FUNCTION_BLOCK FB_AV
VAR_INPUT
END_VAR
VAR_OUTPUT
END_VAR
VAR
	System_Druckluftkompressor_951			: FB_System_DLK_951;
	System_HybriderEnergiespeicher_991		: FB_System_HES_991;
	System_Maschinenversorgung_KW_100		: FB_System_MVKW_100;
	System_Maschinenversorgung_HW_300		: FB_System_MVHW_300;
	System_Haerteofen_961					: FB_System_HO_961;
	System_Maschinenversorgung_WW_245		: FB_System_MVWW_245;
END_VAR
VAR // added by the converter: edge detectors and wires of the graphical bodies
    _w1 : ANY;
END_VAR

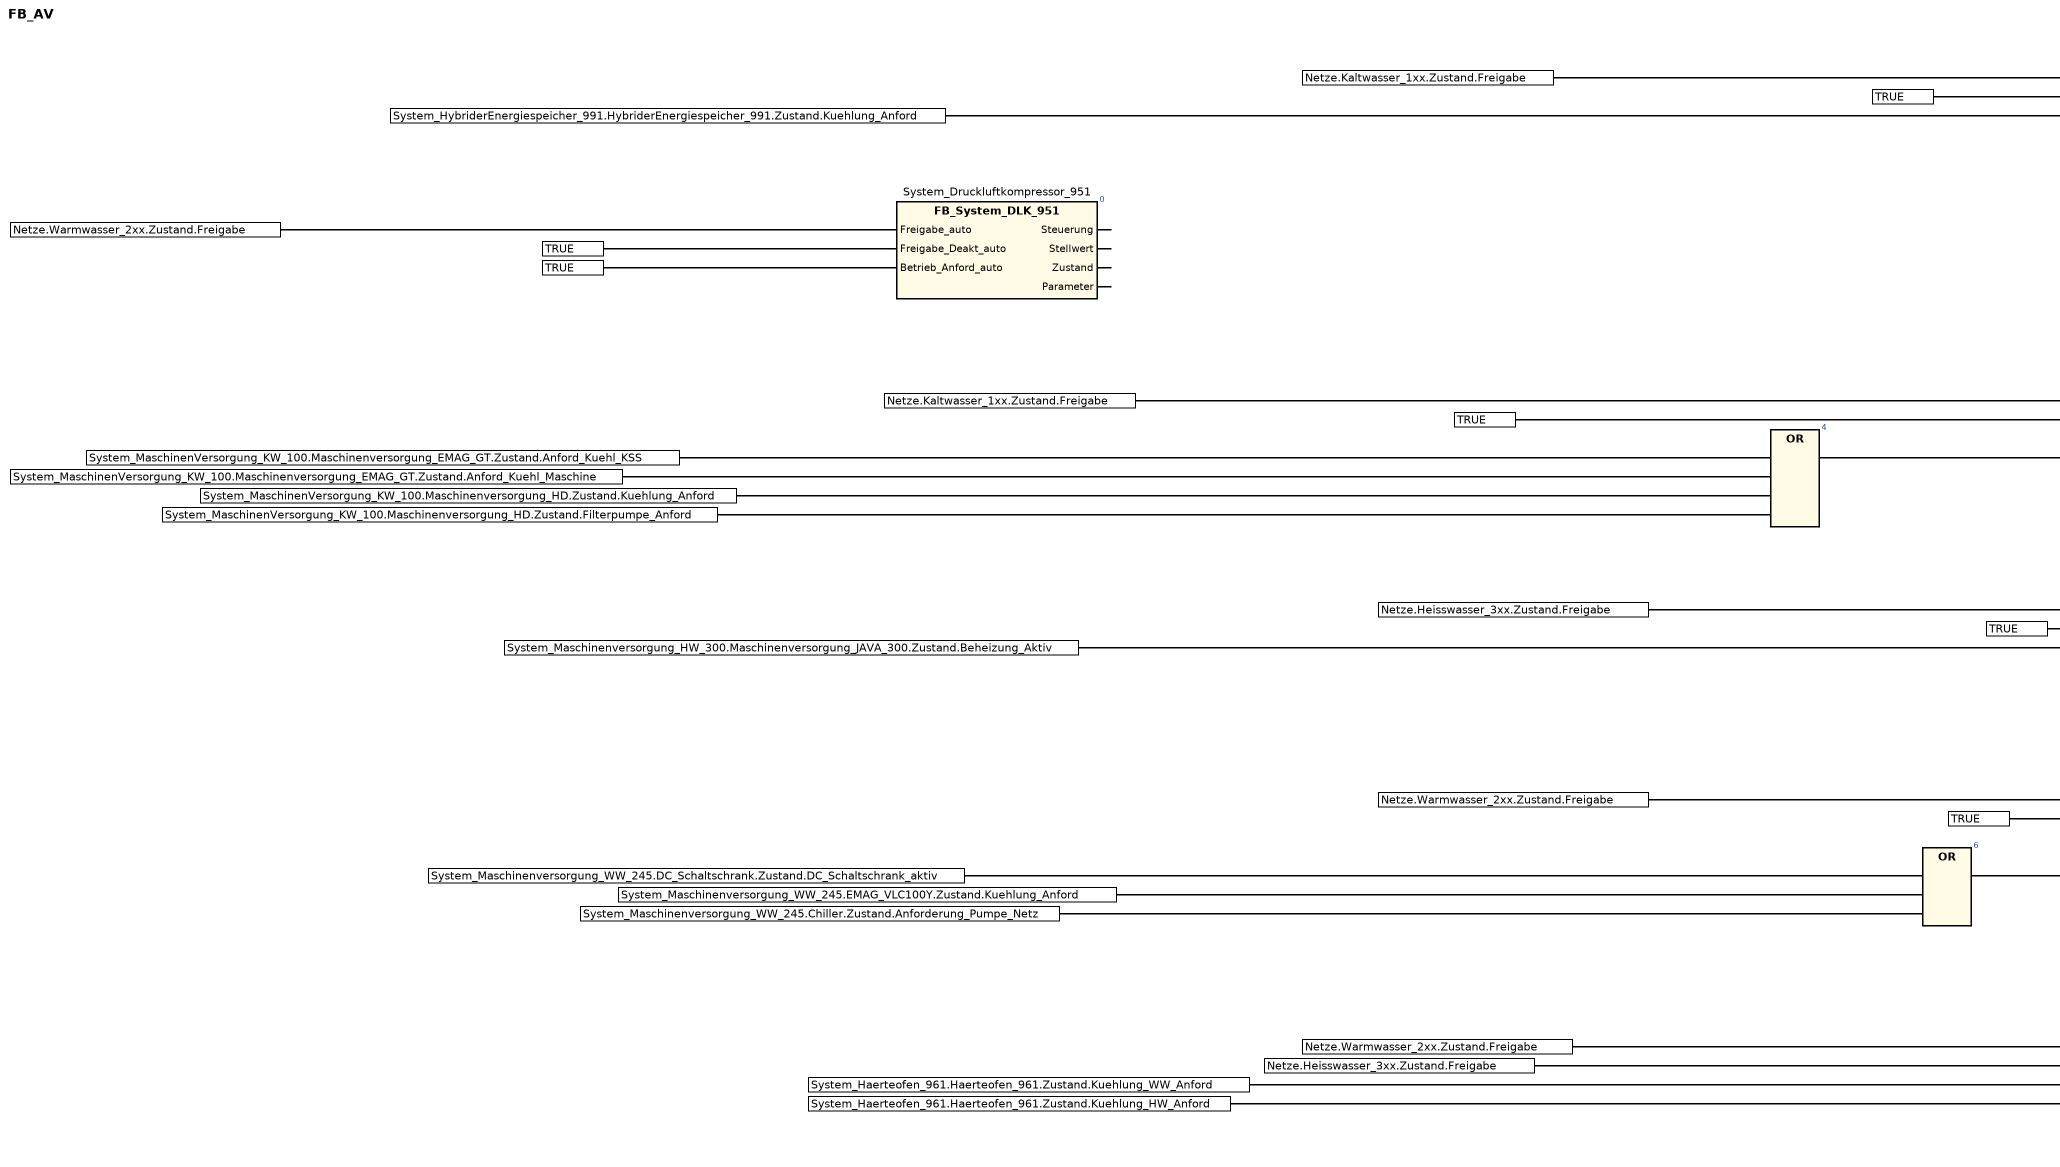
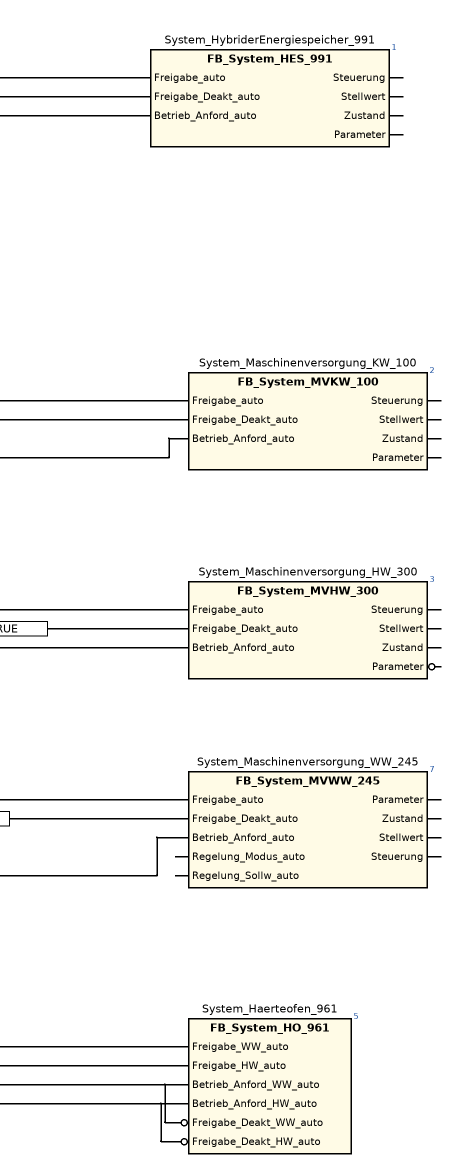
System_Druckluftkompressor_951(
    Freigabe_auto := Netze.Warmwasser_2xx.Zustand.Freigabe,
    Freigabe_Deakt_auto := TRUE,
    Betrieb_Anford_auto := TRUE); // FB_System_DLK_951
System_HybriderEnergiespeicher_991(
    Freigabe_auto := Netze.Kaltwasser_1xx.Zustand.Freigabe,
    Freigabe_Deakt_auto := TRUE,
    Betrieb_Anford_auto := System_HybriderEnergiespeicher_991.HybriderEnergiespeicher_991.Zustand.Kuehlung_Anford); // FB_System_HES_991
System_Maschinenversorgung_KW_100(
    Freigabe_auto := Netze.Kaltwasser_1xx.Zustand.Freigabe,
    Freigabe_Deakt_auto := TRUE,
    Betrieb_Anford_auto := _w1); // FB_System_MVKW_100
System_Maschinenversorgung_HW_300(
    Freigabe_auto := Netze.Heisswasser_3xx.Zustand.Freigabe,
    Freigabe_Deakt_auto := TRUE,
    Betrieb_Anford_auto := System_Maschinenversorgung_HW_300.Maschinenversorgung_JAVA_300.Zustand.Beheizung_Aktiv); // FB_System_MVHW_300
_w1 := System_MaschinenVersorgung_KW_100.Maschinenversorgung_EMAG_GT.Zustand.Anford_Kuehl_KSS OR System_MaschinenVersorgung_KW_100.Maschinenversorgung_EMAG_GT.Zustand.Anford_Kuehl_Maschine OR System_MaschinenVersorgung_KW_100.Maschinenversorgung_HD.Zustand.Kuehlung_Anford OR System_MaschinenVersorgung_KW_100.Maschinenversorgung_HD.Zustand.Filterpumpe_Anford;
System_Haerteofen_961(
    Freigabe_WW_auto := Netze.Warmwasser_2xx.Zustand.Freigabe,
    Freigabe_HW_auto := Netze.Heisswasser_3xx.Zustand.Freigabe,
    Betrieb_Anford_WW_auto := System_Haerteofen_961.Haerteofen_961.Zustand.Kuehlung_WW_Anford,
    Betrieb_Anford_HW_auto := System_Haerteofen_961.Haerteofen_961.Zustand.Kuehlung_HW_Anford,
    Freigabe_Deakt_WW_auto := NOT System_Haerteofen_961.Haerteofen_961.Zustand.Kuehlung_WW_Anford,
    Freigabe_Deakt_HW_auto := NOT System_Haerteofen_961.Haerteofen_961.Zustand.Kuehlung_HW_Anford); // FB_System_HO_961
System_Maschinenversorgung_WW_245(
    Freigabe_auto := Netze.Warmwasser_2xx.Zustand.Freigabe,
    Freigabe_Deakt_auto := TRUE,
    Betrieb_Anford_auto := System_Maschinenversorgung_WW_245.DC_Schaltschrank.Zustand.DC_Schaltschrank_aktiv OR System_Maschinenversorgung_WW_245.EMAG_VLC100Y.Zustand.Kuehlung_Anford OR System_Maschinenversorgung_WW_245.Chiller.Zustand.Anforderung_Pumpe_Netz); // FB_System_MVWW_245

END_FUNCTION_BLOCK

(* stored: Version 1.1.0.1, ProductVersion 3.1.4024.9
   POU FB_AV: Id {dd7bcfbe-cb80-4c01-8582-980d07c39c42}, SpecialFunc None *)
